// TIA Portal V17 export
// export: Created 2022-07-28T18:02:46.2070601Z, ExportSetting None, DisplayName Totally Integrated Automation Portal, DisplayVersion V17, DisplayName TIA Portal Openness, DisplayVersion V17, DisplayName TIA Portal Teamcenter Gateway, DisplayVersion V17, DisplayName TIA Portal Version Control Interface, DisplayVersion V17, DisplayName TIA Portal Test Suite Advanced, DisplayVersion V17, DisplayName SINAMICS Startdrive Advanced, DisplayVersion V17, DisplayName SINAMICS DCC, DisplayVersion V17, DisplayName SINAMICS Startdrive G130, G150, S120, S150, SINAMICS MV, S210, DisplayVersion V17, DisplayName SINAMICS Startdrive G110M, G120, G120C, G120D, G120P, G115D, DisplayVersion V17, DisplayName STEP 7 Professional, DisplayVersion V17, DisplayName SIMATIC Energy Suite, DisplayVersion V17, DisplayName STEP 7 CFC, DisplayVersion V17, DisplayName STEP 7 Safety, DisplayVersion V17, DisplayName WinCC Advanced / Unified PC, DisplayVersion V17, DisplayName SIMATIC Visualization Architect, DisplayVersion V17
FUNCTION_BLOCK "Lib_FB_Timer_OFF_Simple"   // FB12, SCL
{ S7_Optimized_Access := 'TRUE' }
// stored: AutoNumber false, MemoryReserve 100, SetENOAutomatically false
   VAR_INPUT
      IR_CycleTime : Real;   // Last cycle time of PLC, s
      IB_StartTimerInput : Bool;   // 1 = start timer
      IB_ResetTimer : Bool;   // 1 = stop timer. Out = 0
      IR_SpTime : Real;   // Setpoint time for timer, s
   END_VAR
   VAR_OUTPUT
      QB_TimerOut : Bool;   // 1 = timer done
   END_VAR
   VAR
      sR_Cv_ToDone : Real;   // Time to done timer, s
   END_VAR
   VAR_TEMP
      tmp_QB_TimerOut : Bool;
   END_VAR
BEGIN
   //-------------------------------------
   IF #IB_StartTimerInput
   THEN
       #sR_Cv_ToDone := #IR_SpTime;
   END_IF;
   //-------------------------------------
   IF #IB_ResetTimer
   THEN
       #sR_Cv_ToDone := -1.0;
   END_IF;
   //-------------------------------------
   IF NOT #IB_StartTimerInput
       AND #sR_Cv_ToDone > 0
   THEN
       //коли була зміна завдання
       IF #sR_Cv_ToDone >= #IR_SpTime
       THEN
           #sR_Cv_ToDone := #IR_SpTime;
       END_IF;
       //--------------------------------------------
       #sR_Cv_ToDone := #sR_Cv_ToDone - #IR_CycleTime;
   END_IF;
   //--------------------------------------------
   #tmp_QB_TimerOut := #sR_Cv_ToDone > 0
   OR (#IB_StartTimerInput
   AND NOT #IB_ResetTimer);

   #QB_TimerOut := #tmp_QB_TimerOut;
END_FUNCTION_BLOCK
